// TIA Portal project "MesaSeparadora_3" (V14)

(* hardware
DEVICE "S71500/ET200MP station_1"  S7-1500 station
   slot 0: "Rail_0"  Rack  6ES7 590-1***0-0AA0
   slot 1: "PLC_1"  CPU 1516-3 PN/DP  6ES7 516-3AN01-0AB0  V2.1
      slot 3: "CPU display_1"  6ES7591-1BA00-0AA0
   slot 2: "DI 32x24VDC HF_1"  DI 32x24VDC HF  6ES7 521-1BL00-0AB0  V2.1
   slot 3: "DQ 32x24VDC/0.5A HF_1"  DQ 32x24VDC/0.5A HF  6ES7 522-1BL01-0AB0  V1.0
   slot 4: "AI 8xU/I/RTD/TC ST_1"  AI 8xU/I/RTD/TC ST  6ES7 531-7KF00-0AB0  V2.0
   slot 5: "AQ 4xU/I ST_1"  AQ 4xU/I ST  6ES7 532-5HD00-0AB0  V2.0
DEVICE "HMI_1"  KTP700 Basic PN
   slot 0: "KTP700 Basic PN"  KTP700 Basic PN  6AV2 123-2GB03-0AX0  14.0.1.0
   slot 1: "HMI_RT_1"  KTP700 Basic PN  6AV2 123-2GB03-0AX0  14.0.1.0
   slot 5: "HMI_1.IE_CP_1"  PROFINET Interface  14.0.1.0
      slot 1: "PROFINET Interface_1"  PROFINET Interface
         slot 1: "Port_1"  Port
*)

// ===== PLC "PLC_1"  CPU 1516-3 PN/DP =====

VAR_GLOBAL   // PLC tag table "Default tag table"
   "altura_gra" AT %I0.0 : Bool;
   "altura_med" AT %I0.1 : Bool;
   "altura_peq" AT %I0.2 : Bool;
   "queda1" AT %I0.3 : Bool;
   "queda2" AT %I0.4 : Bool;
   "queda3" AT %I0.5 : Bool;
   "valv_solen_1_re" AT %Q0.1 : Bool;
   "valv_solen_2" AT %Q0.2 : Bool;
   "valv_solen_3" AT %Q0.3 : Bool;
   "motor" AT %Q0.4 : Bool;
   "valv_solen_1_av" AT %Q0.0 : Bool;
   "mem_altura_gra" AT %M0.0 : Bool;
   "mem_altura_med" AT %M0.1 : Bool;
   "mem_altura_peq" AT %M0.2 : Bool;
   "mem_indutivo" AT %M0.3 : Bool;
   "capacitivo" AT %I0.6 : Bool;
   "indutivo" AT %I0.7 : Bool;
   "bot_liga_deslig_est" AT %M0.4 : Bool;
   "mem_capacitvo" AT %M0.5 : Bool;
   "mem_valv_solen_1_av" AT %M0.6 : Bool;
   "mem_valv_solen_2_re" AT %M0.7 : Bool;
   "bob_aux_1" AT %M1.0 : Bool;
   "box_aux_2" AT %M1.1 : Bool;
   "box_aux_3" AT %M1.2 : Bool;
   "bob_aux_4" AT %M1.3 : Bool;
   "cv_ctu_pc_plast" AT %MW20 : Word;
   "cv_ctu_pc_met_g" AT %MW22 : Word;
   "cv_ctu_pc_met_m" AT %MW24 : Word;
   "cv_ctu_pc_met_p" AT %MW26 : Word;
   "sens_fim_curso" AT %I1.0 : Bool;
   "reset" AT %M1.4 : Bool;
END_VAR

// folder: System blocks/Program resources

DATA_BLOCK "CTU_PC_PLAST"   // DB1
{ S7_Optimized_Access := 'TRUE' }
AUTHOR : Simatic
FAMILY : IEC
NAME : CNTR
VERSION : 1.0
// stored: InstanceOfName IEC_COUNTER
"IEC_COUNTER"
BEGIN
END_DATA_BLOCK

DATA_BLOCK "CTU_PC_MET_P"   // DB2
{ S7_Optimized_Access := 'TRUE' }
AUTHOR : Simatic
FAMILY : IEC
NAME : CNTR
VERSION : 1.0
// stored: InstanceOfName IEC_COUNTER
"IEC_COUNTER"
BEGIN
END_DATA_BLOCK

DATA_BLOCK "CTU_PC_MET_M"   // DB3
{ S7_Optimized_Access := 'TRUE' }
AUTHOR : Simatic
FAMILY : IEC
NAME : CNTR
VERSION : 1.0
// stored: InstanceOfName IEC_COUNTER
"IEC_COUNTER"
BEGIN
END_DATA_BLOCK

DATA_BLOCK "CTU_PC_MET_G"   // DB4
{ S7_Optimized_Access := 'TRUE' }
AUTHOR : Simatic
FAMILY : IEC
NAME : CNTR
VERSION : 1.0
// stored: InstanceOfName IEC_COUNTER
"IEC_COUNTER"
BEGIN
END_DATA_BLOCK

// folder: (top level)

ORGANIZATION_BLOCK "Main"   // OB1, LAD, ProgramCycle
TITLE = "Programa Principal"
{ S7_Optimized_Access := 'TRUE' }
VERSION : 0.1
   VAR_INPUT
      Initial_Call : Bool;   // Initial call of this OB
      Remanence : Bool;   // =True, if remanent data are available
   END_VAR
BEGIN

REGION Network 1: Lógica para ligar/desligar o motor manualmente
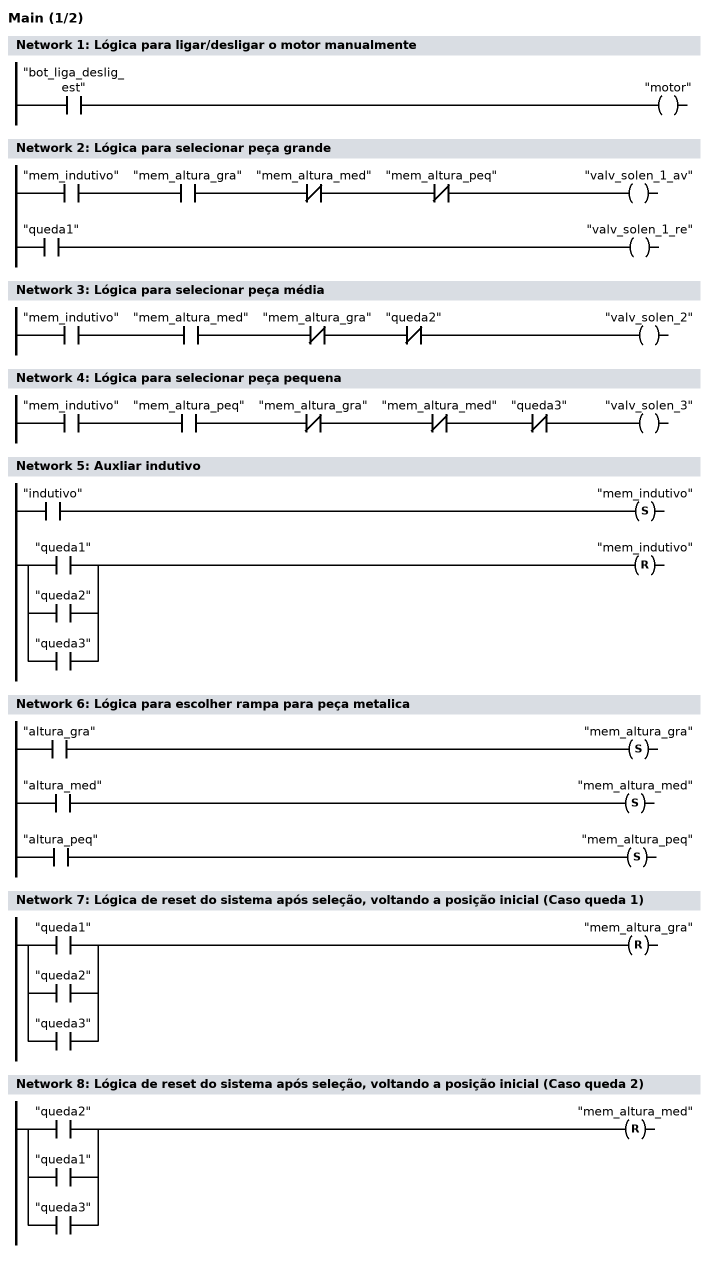
   RUNG wire#powerrail
      Contact( "bot_liga_deslig_est" )
      Coil( "motor" )
   END_RUNG
   // the same network as SCL:
   "motor" := "bot_liga_deslig_est";
END_REGION

REGION Network 2: Lógica para selecionar peça grande
   RUNG wire#powerrail
      Contact( "mem_indutivo" )
      Contact( "mem_altura_gra" )
      I_Contact( "mem_altura_med" )
      I_Contact( "mem_altura_peq" )
      Coil( "valv_solen_1_av" )
   END_RUNG
   RUNG wire#powerrail
      Contact( "queda1" )
      Coil( "valv_solen_1_re" )
   END_RUNG
   // the same network as SCL:
   "valv_solen_1_av" := "mem_indutivo" AND "mem_altura_gra" AND NOT "mem_altura_med" AND NOT "mem_altura_peq";
   "valv_solen_1_re" := "queda1";
END_REGION

REGION Network 3: Lógica para selecionar peça média
   RUNG wire#powerrail
      Contact( "mem_indutivo" )
      Contact( "mem_altura_med" )
      I_Contact( "mem_altura_gra" )
      I_Contact( "queda2" )
      Coil( "valv_solen_2" )
   END_RUNG
   // the same network as SCL:
   "valv_solen_2" := "mem_indutivo" AND "mem_altura_med" AND NOT "mem_altura_gra" AND NOT "queda2";
END_REGION

REGION Network 4: Lógica para selecionar peça pequena
   RUNG wire#powerrail
      Contact( "mem_indutivo" )
      Contact( "mem_altura_peq" )
      I_Contact( "mem_altura_gra" )
      I_Contact( "mem_altura_med" )
      I_Contact( "queda3" )
      Coil( "valv_solen_3" )
   END_RUNG
   // the same network as SCL:
   "valv_solen_3" := "mem_indutivo" AND "mem_altura_peq" AND NOT "mem_altura_gra" AND NOT "mem_altura_med" AND NOT "queda3";
END_REGION

REGION Network 5: Auxliar indutivo
   RUNG wire#powerrail
      Contact( "indutivo" )
      S_Coil( "mem_indutivo" )
   END_RUNG
   RUNG wire#powerrail
      Contact( "queda1" )
      wire#w1
      R_Coil( "mem_indutivo" )
   END_RUNG
   RUNG wire#powerrail
      Contact( "queda2" )
   END_RUNG wire#w1
   RUNG wire#powerrail
      Contact( "queda3" )
   END_RUNG wire#w1
   // the same network as SCL:
   IF "indutivo" THEN "mem_indutivo" := TRUE; END_IF;
   IF "queda1" OR "queda2" OR "queda3" THEN "mem_indutivo" := FALSE; END_IF;
END_REGION

REGION Network 6: Lógica para escolher rampa para peça metalica
   RUNG wire#powerrail
      Contact( "altura_gra" )
      S_Coil( "mem_altura_gra" )
   END_RUNG
   RUNG wire#powerrail
      Contact( "altura_med" )
      S_Coil( "mem_altura_med" )
   END_RUNG
   RUNG wire#powerrail
      Contact( "altura_peq" )
      S_Coil( "mem_altura_peq" )
   END_RUNG
   // the same network as SCL:
   IF "altura_gra" THEN "mem_altura_gra" := TRUE; END_IF;
   IF "altura_med" THEN "mem_altura_med" := TRUE; END_IF;
   IF "altura_peq" THEN "mem_altura_peq" := TRUE; END_IF;
END_REGION

REGION Network 7: Lógica de reset do sistema após seleção, voltando a posição inicial (Caso queda 1)
   RUNG wire#powerrail
      Contact( "queda1" )
      wire#w1
      R_Coil( "mem_altura_gra" )
   END_RUNG
   RUNG wire#powerrail
      Contact( "queda2" )
   END_RUNG wire#w1
   RUNG wire#powerrail
      Contact( "queda3" )
   END_RUNG wire#w1
   // the same network as SCL:
   IF "queda1" OR "queda2" OR "queda3" THEN "mem_altura_gra" := FALSE; END_IF;
END_REGION

REGION Network 8: Lógica de reset do sistema após seleção, voltando a posição inicial (Caso queda 2)
   RUNG wire#powerrail
      Contact( "queda2" )
      wire#w1
      R_Coil( "mem_altura_med" )
   END_RUNG
   RUNG wire#powerrail
      Contact( "queda1" )
   END_RUNG wire#w1
   RUNG wire#powerrail
      Contact( "queda3" )
   END_RUNG wire#w1
   // the same network as SCL:
   IF "queda2" OR "queda1" OR "queda3" THEN "mem_altura_med" := FALSE; END_IF;
END_REGION

REGION Network 9: Lógica de reset do sistema após seleção, voltando a posição inicial (Caso queda 3)
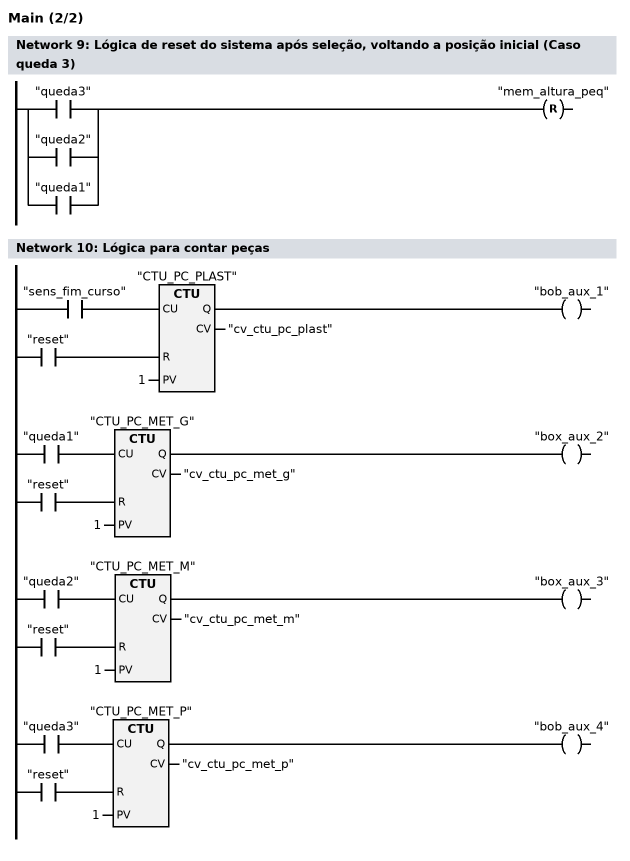
   RUNG wire#powerrail
      Contact( "queda3" )
      wire#w1
      R_Coil( "mem_altura_peq" )
   END_RUNG
   RUNG wire#powerrail
      Contact( "queda2" )
   END_RUNG wire#w1
   RUNG wire#powerrail
      Contact( "queda1" )
   END_RUNG wire#w1
   // the same network as SCL:
   IF "queda3" OR "queda2" OR "queda1" THEN "mem_altura_peq" := FALSE; END_IF;
END_REGION

REGION Network 10: Lógica para contar peças
   "CTU_PC_PLAST".CTU(CU := "sens_fim_curso", R := "reset", PV := 1, CV => "cv_ctu_pc_plast");
   "bob_aux_1" := "CTU_PC_PLAST".Q;
   "CTU_PC_MET_G".CTU(CU := "queda1", R := "reset", PV := 1, CV => "cv_ctu_pc_met_g");
   "box_aux_2" := "CTU_PC_MET_G".Q;
   "CTU_PC_MET_M".CTU(CU := "queda2", R := "reset", PV := 1, CV => "cv_ctu_pc_met_m");
   "box_aux_3" := "CTU_PC_MET_M".Q;
   "CTU_PC_MET_P".CTU(CU := "queda3", R := "reset", PV := 1, CV => "cv_ctu_pc_met_p");
   "bob_aux_4" := "CTU_PC_MET_P".Q;
END_REGION
END_ORGANIZATION_BLOCK

(* ===== HMI "HMI_RT_1" =====
system functions are stored by id; their names below are inferred from use
connection "HMI_Connection_1": ETHERNET, SMART_S7_1500_OMS

HMI tags "Default tag table"
   "Tag_ScreenNumber" : UInt, internal
   "altura_peq" : Bool = PLC altura_gra AT %I0.0, 1 s
   "altura_med" : Bool = PLC altura_med AT %I0.1, 1 s
   "altura_gra" : Bool = PLC altura_peq AT %I0.2, 1 s
   "queda1" : Bool = PLC queda1 AT %I0.3, 1 s
   "queda2" : Bool = PLC queda2 AT %I0.4, 1 s
   "queda3" : Bool = PLC queda3 AT %I0.5, 1 s
   "bot_liga_deslig_est" : Bool = PLC bot_liga_deslig_est AT %M0.4, 1 s
   "valv_solen_1_av" : Bool = PLC valv_solen_1_av AT %Q0.0, 1 s
   "valv_solen_1_re" : Bool = PLC valv_solen_1_re AT %Q0.1, 1 s
   "cv_ctu_pc_plast" : Word = PLC cv_ctu_pc_plast AT %MW20, 1 s
   "cv_ctu_pc_met_m" : Word = PLC cv_ctu_pc_met_m AT %MW24, 1 s
   "cv_ctu_pc_met_g" : Word = PLC cv_ctu_pc_met_g AT %MW22, 1 s
   "cv_ctu_pc_met_p" : Word = PLC cv_ctu_pc_met_p AT %MW26, 1 s
   "reset" : Bool = PLC reset AT %M1.4, 1 s

Template "Template_1" 800x480
   Button "Exit" at 714,429 size 71x50; TextOff 'Exit'; PictureOff "ExitRuntime_KTP700_Basic_PN_TR"; PictureOn "ExitRuntime_KTP700_Basic_PN_TR"
      on Release: StopRuntime(0)
   Button "Template_Button" at 614,429 size 71x50; TextOff 'Text'
   Button "Template_Button_1" at 514,429 size 71x50; TextOff 'Text'
   Button "Template_Button_2" at 414,429 size 71x50; TextOff 'Text'
   Button "Template_Button_3" at 314,429 size 71x50; TextOff 'Text'
   Button "Template_Button_4" at 214,429 size 71x50; TextOff 'Text'
   Button "Alarms" at 114,429 size 71x50; TextOff 'Alarms'; PictureOff "AlarmDisplay_KTP700_Basic_PN_TR"; PictureOn "AlarmDisplay_KTP700_Basic_PN_TR"
      on Release: function_ef3f5d25("Alarm window_Unacknowledged", -1)
   Button "Start screen" at 14,429 size 71x50; TextOff 'Start screen'; PictureOff "NavigateHome_KTP700_Basic_PN_TR"; PictureOn "NavigateHome_KTP700_Basic_PN_TR"
      on Release: ActivateScreen("Root screen", 0)
   SymbolicIOField "Symbolic_IO_Field_Screen" at 93,9 size 600x33; TextOff '0'; TextOn '1'; TextList "TextList_ScreenNames"
      ProcessValue <- "Tag_ScreenNumber"
      on Change: ActivateScreenByNumber("Tag_ScreenNumber", 0)
   DateTimeField "HmiScreenItemData" at 695,25 size 105x25
   DateTimeField "HmiScreenItemData_1" at 695,0 size 105x25
   GraphicView "Logo" at 0,0 size 91x51; Picture "Logo of HMI_1"

screen "Root screen" 800x480, template "Template_1"
   on GenerateScreen: SetTag("Tag_ScreenNumber", 1)
   Button "Button_1" at 33,77 size 132x52; TextOff 'Ligar Motor'
      on Press: InvertBit("bot_liga_deslig_est")
   IOField "I/O field_2" at 172,211 size 124x50; FormatPattern 99999
      ProcessValue <- "cv_ctu_pc_met_m"
   IOField "I/O field_4" at 172,337 size 124x50; FormatPattern 99999
      ProcessValue <- "cv_ctu_pc_plast"
   TextField "Text field_7" at 311,347 size 210x23; Text 'Qtd. Peças Não Metálicas'
   TextField "Text field_8" at 311,224 size 235x23; Text 'Qtd. Peças Metálicas Médias'
   TextField "Text field_9" at 311,285 size 257x23; Text 'Qtd. Peças Metálicas Pequenas'
   TextField "Text field_10" at 311,161 size 245x23; Text 'Qtd. Peças Metálicas Grandes'
   Button "Button_2" at 627,358 size 132x52; TextOff 'Reset'
      on Press: function_b14e0dd5("reset", 0)
   IOField "I/O field_1" at 172,148 size 124x50; FormatPattern 99999
      ProcessValue <- "cv_ctu_pc_met_g"
   IOField "I/O field_3" at 172,273 size 124x50; FormatPattern 99999
      ProcessValue <- "cv_ctu_pc_met_p"

screen "System screens" 800x480, template "Template_1"
   on GenerateScreen: SetTag("Tag_ScreenNumber", 2)
   Button "Back" at 1,52 size 159x47; TextOff 'Back'
      on Release: ActivateScreen("Root screen", 0)
   Button "HmiScreenItemData" at 36,146 size 159x47; TextOff 'Project information'; PictureOff "Navigates to Project information for KTP700 Basic+ PN 14.0.1.0"; PictureOn "Navigates to Project information for KTP700 Basic+ PN 14.0.1.0"
      on Release: ActivateScreen("Project information", 0)

screen "Project information" 800x480, template "Template_1"
   on GenerateScreen: SetTag("Tag_ScreenNumber", 3)
   TextField "HmiScreenItemData" at 35,102 size 171x28; Text 'Project name:'
   TextField "HmiScreenItemData_1" at 241,102 size 524x28; Text 'MesaSeparadora'
   TextField "HmiScreenItemData_2" at 35,132 size 171x28; Text 'Created on:'
   TextField "HmiScreenItemData_3" at 241,132 size 524x28; Text '3/22/2024 4:47:41 PM'
   TextField "HmiScreenItemData_4" at 35,162 size 171x28; Text 'Author:'
   TextField "HmiScreenItemData_5" at 241,162 size 524x28; Text 'Aluno'
   TextField "HmiScreenItemData_6" at 35,192 size 171x28; Text 'Description:'
   TextField "HmiScreenItemData_7" at 241,192 size 524x28; Text '(not configured)'
   Button "Back" at 1,52 size 159x47; TextOff 'Back'
      on Release: ActivateScreen("System screens", 0)
*)